FUNCTION_BLOCK FB_PrintModule_WEU EXTENDS FB_PrintModule_Base
VAR_INPUT
  fPUPlate1_Temperature : LREAL;  // PU Plate1 temperature
  fPUPlate2_Temperature : LREAL;  // PU Plate2 temperature
END_VAR
VAR
  (* Module specific sub-modules - WEU module contains a 
    - print position (encoder input to print domain translation)
    - Mark sensor with a mark detection module which provices a camera trigger and start position detection
    - Mark definition (used by the detection and camera)
  *)
  fbPrintPosition    : FB_PrintPositionDmax;   // a position per pm (external encoder wheel)
  fbMarkCameraWeu    : FB_MarkCamera_WEU;      // Mark detection camera
  
  // sync CT trigger with Camera detection
  _bNewCT             : BOOL;   // a new ct is received to be treated
  _iNewCT             : I_CT;   // new ct to be treated
  _bNewStartPosX0     : BOOL;   // a new startpos detected by cam
  _nNewStartPosX0     : DINT;   // new startpos X0 deteced by cam
  
  fbEncoderResoDetect : FB_EffectiveEncoderResolutionDetection;     // Effective encoder resolution detection
  fbFineAlignement    : FB_FineAlignement;     // additional grid corrections, PU Deformation/correction (4p, banana, ...)

  // messages specific
  fbMsgWeu            : ARRAY[1..nC_NumMsgWeu] OF FB_MESSAGE;  (*Messages*)
  
  // view
  fbView              : FB_PrintModule_WEU_View;    // additional controls for print module visus
END_VAR
VAR CONSTANT
  nC_NumMsgWeu        : UDINT := 6;           // number of internal messages
END_VAR

IF NOT bInit THEN RETURN; END_IF

// position
fbPrintPosition.fEnoderResolution := _pModuleMachineState^.fEncoderResolution;    // encoder resolution from machine
fbPrintPosition();

// -------------------------
// StartTrigger evaluation -> apply new CT to Tracking (created from CTM externally)
// Synchronize CT (EvPos) received from CTManger (Main) to the local StartTrigger detection and positioning
// -- reset triggers if not active
IF NOT bReadyForPrinting THEN
  _bNewCT := 0; _bNewStartPosX0 := 0;
END_IF
// -- new StartTrigger (X0)
IF bReadyForPrinting AND _iStartPos.bStartTrig AND _iStartPos.bValid THEN
  // buffer/save new start trigger
  _bNewStartPosX0 := TRUE;
  _nNewStartPosX0 := _iStartPos.nStartPositionX0;      // save detected start position for next CT to be applied to this module¨
  
  LogLvl(Lvl:=E_LogSeverity.Debug, Msg:=F_Concat3(
    F_Concat2(_pModuleSetup^.aName, ' New StartTrigger detected:'),
    F_Concat2(' at position X0:', TO_STRING(_nNewStartPosX0)),
    F_Concat2(' PM is now at: ', TO_STRING(fbPrintPosition.getPosition())),
  ));
  
  IF _bNewCT THEN   // we have an attached CT
      LogLvl(Lvl:=E_LogSeverity.Debug, Msg:=F_Concat3(
      F_Concat2(_pModuleSetup^.aName, ' Track NewCT:'),
      F_Concat2(' internal (print)Pos X0:', TO_STRING(_nNewStartPosX0)),
      F_Concat2(' with CT:', _iNewCT.print(0))
    ));
    
    _iNewCT.nPosPrint_X0 := _nNewStartPosX0;                        // set print pos to new dected in this module position domain
    fbCTTracker.RegisterCT(iCT:=_iNewCT, nX0:=_nNewStartPosX0);     // register ct for tracking in modules position and tracking system
  ELSE
    // spurious trigger (CTs not yet arrived at PMx, but receive some StartTriggers
    LogLvl(Lvl:=E_LogSeverity.Debug, Msg:=F_Concat3('StartTrigger at Pos X0:', TO_STRING(_nNewStartPosX0), ' but no CT received'));
	END_IF
  
  // reset internals (saved triggers)
  _bNewCT := FALSE; _iNewCT := 0; 
  _bNewStartPosX0 := FALSE;
END_IF

// Camera (is per module)
fbMarkCameraWeu(
  bReadyForPrinting   := bReadyForPrinting,
  nCurrentPosition    := _iPrintPosition.getPosition(),
  fCurrentSpeed       :=_iPrintPosition.getSpeed(),
  bPrintMarkExist     :=_pModuleMachineState^.bPrintMarkExist,
  bPrintDirReverse    :=_pModuleMachineState^.bPrintDirection,
  nUsePerRepeatInLine :=SEL(_pModuleMachineState^.nUsePerRepeatInLine=0, _pModuleMachineState^.nUsePerRepeatInLine, 1),
  fMarkSizeDefault    :=_pModuleMachineState^.fMarkBaseSize,
  fMarkDistRepeatToStartMark := _pModuleMachineState^.fMarkDistToStartMark,
  fMarkDistFromCenter := _pModuleMachineState^.fMarkToPrintdataCenterY
);

// Effective Encoder detection - Neutral fibre calculation with additional mark sensors
fbEncoderResoDetect(
  //bIKp_MarkTrigger01:=,
  //tIKp_TimeStampPos01:=,
  //tIKn_TimeStampNeg01:=,
  //bIKp_MarkTrigger02:=,
  //tIKp_TimeStampPos02:=,
  //tIKn_TimeStampNeg02:=,
  nPulse:=TO_DINT(fbPrintPosition.IlEncoderPulse),
  fCurrentResolution:=_pModuleMachineState^.fEncoderResolution,
  fEncoderPulseDistMin:=_pModuleMachineState^.fEncoderDetectPulseMin,
  fEncoderPulseDistMax:=_pModuleMachineState^.fEncoderDetectPulseMax,
  nDisInPulseFilterSz:=_pModuleMachineState^.nEncoderDetectFilterSz,
  fMinMarkLength:=(0.5 - 0.1) * _pModuleMachineState^.fMarkBaseSize * 1_000_000,  // 0.5*a (0*a from triangle)
  fMaxMarkLength:=(  3 + 0.1) * _pModuleMachineState^.fMarkBaseSize * 1_000_000,  //   2*a (1*a from triangle) 
  // --> the following would only work when teached
  //fMinMarkLength:=fbMarkCameraWeu.pFbMarkDefinition^.fMinMarkLength - fbMarkCameraWeu.pFbMarkDefinition^.fMarkLengthMargin * 1_000_000,
  //fMaxMarkLength:=fbMarkCameraWeu.pFbMarkDefinition^.fMaxMarkLength + fbMarkCameraWeu.pFbMarkDefinition^.fMarkLengthMargin * 1_000_000,
  //bUpdate=>,
  fDisInPulse=>_pModuleMachineFeedback^.fEncoderStepsMeasured
);

(*PU corrections*)
IF GVL_Deformation.bC_UsePUDeformation THEN
  fbFineAlignement.fT_PL1 := fPUPlate1_Temperature;
  fbFineAlignement.fT_PL2 := fPUPlate2_Temperature;
  fbFineAlignement();
END_IF

fbView();

// call module base
SUPER^();

// messages print module
fbMsgWeu[ 1](bI_Status := bTestMsg OR fbMarkCameraWeu.bMissingMarks);
fbMsgWeu[ 2](bI_Status := bTestMsg OR _pModuleMachineState^.bDriftControlMissMarks);
fbMsgWeu[ 3](bI_Status := bTestMsg OR fbMarkCameraWeu.bMarkDetectionErrors);
fbMsgWeu[ 4](bI_Status := bTestMsg OR fbMarkCameraWeu.bTeachError);
fbMsgWeu[ 5](bI_Status := bTestMsg OR fbMarkCameraWeu.bImageLengthInvalid);
fbMsgWeu[ 6](bI_Status := bTestMsg OR _bGridLimited);

IF fb_MsgQueue.bO_ReceiptMessage THEN
  fbMarkCameraWeu.ackErrors();
  _bGridLimited := FALSE;
END_IF

// simulation
SimUpdate();

PROPERTY bForceNoCorrectionButYShiftMode : BOOL
SET
FOR nCtr := 1 TO GVL_WEU.nC_MaxWorkerPrintPerPm DO
  fbWorkerPrint[nCtr].bForceNoCorrectionButShiftMode := bForceNoCorrectionButYShiftMode;
END_FOR
END_SET
END_PROPERTY

METHOD Init : BOOL
VAR_INPUT
  pModulesSetup         : POINTER TO ST_CassetteSetup;          // Module Setup Settings
  pAdsSa                : POINTER TO FB_ADS_DVTSHEETALIGNMENT;  // ADS sheet alignement
  pAdsCam               : POINTER TO FB_ADS_CAMERA;             // ADS camera
  pAdsParent            : POINTER TO FB_ADS_Config;             // Parent ADS config reference (Parent ADS block and module ref)

  // config print
  fCycleTime            : LREAL;                // task cycle time in [s]
  fPrintUnitWidth       : LREAL;                // PrintUnit width mechanical [m]
  // references
  iModule               : I_Module;             // system status interface (for sleep, estop, ...), may shadow states from machine inputs
  iPrintGlobal          : I_PrintGlobal;        // interface for module to master (main) communication
  pMachineInputs        : POINTER TO ST_ModuleMachineInterface_IN;
  pMachineOutputs       : POINTER TO ST_ModuleMachineInterface_OUT;
END_VAR
VAR
  nCtr : UDINT;
END_VAR
// Parameter checks
IF pModulesSetup = 0 OR pAdsSa = 0 OR pAdsCam = 0 OR 
    pMachineInputs = 0 OR pMachineOutputs = 0 THEN
    // set here from local fb instances: OR iModuleMaster = 0 OR iPosition = 0 OR iStartPos = 0 THEN
  LogError('init(): Invalid parameter');
  RETURN;
END_IF

// position
fbPrintPosition.Init(fPrintResolution:=pModulesSetup^.pSetupPrint^.nPrintResolution, fSubPxResolution:=pModulesSetup^.pSetupPrint^.nSubPixelResolution, fTaskCycleTime:=fCycleTime);
_iPrintPosition := fbPrintPosition;  // select reference position

// -- Mark camera
fbMarkCameraWeu.InitMarkCamera(
  fPrintUnitResolution:=_iPrintPosition.fPrintResolution, 
  fPrintUnitSubPx:=_iPrintPosition.fSubPxResolution
);
fbMarkCameraWeu.sVisuName := 'VISU_MarkCamera_WEU';
fbWorkerCamera.RegisterCamera(fbMarkCameraWeu);

// -- Sheet/Camera trigger & mark detection
_iStartPos := fbMarkCameraWeu.fbMarkDetection;  // select start position detection

SUPER^.Init(
  pModulesSetup     := pModulesSetup,
  pAdsSa            := pAdsSa,
  pAdsCam           := pAdsCam,
  pAdsParent        := pAdsParent,
  // config print
  fCycleTime        := fCycleTime,
  fPrintUnitWidth   := fPrintUnitWidth,
  // references     
  iPrintGlobal      := iPrintGlobal,     // internal subm
  iModule           := iModule, 
  pMachineInputs    := pMachineInputs,
  pMachineOutputs   := pMachineOutputs
);

// Effective Encoder Resolution detection (NeutralFibre correction)
fbEncoderResoDetect.Init();

// additional grid point corrections
fbFineAlignement.init(pAdsCam := pAdsCam, fPxReso := _iPrintPosition.fPrintResolution, fPuWidth := fPrintUnitWidth);
// - register them to workers
FOR nCtr := 1 TO GVL_WEU.nC_MaxWorkerPrintPerPm DO
  fbWorkerPrint[nCtr].RegisterGridCorrection(iGridCorrection:=fbFineAlignement);
END_FOR 

fbView.init(pModule:=THIS, pPositioning:=ADR(fbPrintPosition));
setLogLevels(lvl:=E_LogSeverity.Info);

FOR nCtr := 1 TO nC_NumMsgWeu DO
  fbMsgWeu[nCtr].pI_MsgConfig       := ADR(sL_MsgConfig);
  fbMsgWeu[nCtr].iI_MsgLocation     := 1;
END_FOR;
fbMsgWeu[ 1].iI_MsgNumber      := eCPr_PrintMarkError_Generic;        // mark detection error
fbMsgWeu[ 2].iI_MsgNumber      := eCMa_DRIFT_CONTR_ERROR;             // drift controller error
fbMsgWeu[ 3].iI_MsgNumber      := eCPr_SHEET_MARK_DETECTION;          // mark error missing/faulty
fbMsgWeu[ 4].iI_MsgNumber      := eC_STAG_CAM_TEACH_ERROR;            // teach error
fbMsgWeu[ 5].iI_MsgNumber      := eC_STAG_IMAGELENGTH_NOT_SUPPORTED;  // image length not supported (out of supported range)
fbMsgWeu[ 6].iI_MsgNumber      := eC_STAG_DEFORMATION_LIMITED;        // deformation calculated was limited to min/max before sending

Init := bInit;   // set in the SUPER class
END_METHOD

PROPERTY pMsgConfig : POINTER TO ST_MSG_CONFIG
GET
pMsgConfig := ADR(sL_MsgConfig);
END_GET
END_PROPERTY

METHOD PROTECTED setLogLevels
VAR_INPUT
  lvl : E_LogSeverity;
END_VAR
// - fb itself
LogLevel := lvl;
// - base
SUPER^.setLogLevels(lvl:=lvl);
// - weu
fbPrintPosition.LogLevel := lvl;
fbMarkCameraWeu.LogLevel := lvl;
END_METHOD

METHOD PRIVATE SimUpdate
VAR_INPUT
END_VAR
VAR_INST
  rfTrig_SimEnable : RF_TRIG;
  
  //parameter backup
  fCamMark_ToPrint, fCamMark_toDetect : LREAL;
  fCamNo_ToPrint, fCamNo_toDetect : LREAL;
END_VAR
rfTrig_SimEnable(CLK:=fbSim.bSimEnable);
IF    rfTrig_SimEnable.RT THEN
  // ev. enable
  //fbWorkerCamera.bWorkerEnable := TRUE;
  //fbWorkerDeformation.bWorkerEnable := TRUE;
  //fbWorkerPrint[1].bWorkerEnable := TRUE;
  //fbWorkerPrint[2].bWorkerEnable := TRUE;
  
  fbPrintPosition.bSimEnable  := TRUE;
  fbMarkCameraWeu.bSimulate := TRUE;

  // set some working config values
  // -backup original
  fCamMark_ToPrint  := fbMarkCameraWeu.fCameraToPrintOffset;
  fCamMark_toDetect := fbMarkCameraWeu.fDetectToCameraOffset;
  // -set sim val
  fbMarkCameraWeu.fCameraToPrintOffset := 0.4;
  fbMarkCameraWeu.fDetectToCameraOffset := 0.01;
  
  
ELSIF rfTrig_SimEnable.FT THEN
  // ev. disable
  fbPrintPosition.bSimEnable  := FALSE;
  fbMarkCameraWeu.bSimulate := FALSE;

  fbMarkCameraWeu.fCameraToPrintOffset := fCamMark_ToPrint;
  fbMarkCameraWeu.fDetectToCameraOffset := fCamMark_toDetect;
  
ELSIF fbSim.bSimEnable THEN
  // enabled
  ;
ELSE
  ; // disabled
END_IF
END_METHOD

(*
  Container triggered at position - callback.
*)
METHOD trigger : BOOL
VAR_INPUT
	sEvPos	: ST_PositionEventData;
END_VAR
IF NOT bInit THEN RETURN; END_IF
IF sEvPos.iCT = 0 THEN RETURN; END_IF


// buffer new ct
_bNewCT := TRUE;
_iNewCT := sEvPos.iCT;

LogLvl(Lvl:=E_LogSeverity.Debug, Msg:=F_Concat3(
  F_Concat2(_pModuleSetup^.aName, ' NewCT PosEv:'),
  F_Concat2(' at (Main)TrackPos:', TO_STRING(sEvPos.nTrigPos)),
  F_Concat2(' with CT:', sEvPos.iCT.print(0))
));
END_METHOD

END_FUNCTION_BLOCK

(* stored: Version 1.1.0.1, ProductVersion 3.1.4024.11
   POU FB_PrintModule_WEU: Id {bf81d19f-9fa7-4acb-8cca-087a288b3f4d}, SpecialFunc None
   Folder I_PositionEvent_ovrd: Id {212612fd-c98f-4fcb-8ea9-fac5585d1647}
   Folder Simulation: Id {ff45cf45-269f-4fec-ab1d-0aca9951a18d}
   Property bForceNoCorrectionButYShiftMode: Id {b65a9350-831c-45ea-8f78-0fa9026ef73e}
   Set Set: Id {3d096227-cb0c-4e6c-ae20-0ca9a6fd3412}
   Method Init: Id {fba0a279-e9f9-46b1-8f8f-0e7a0e308a34}
   Property pMsgConfig: Id {3f9ad2f8-f49c-46e8-8c7b-162fe18749a6}
   Get Get: Id {5bcaf950-0c98-4a16-8209-bb10ff6fbca0}
   Method setLogLevels: Id {e26383c7-5f29-468c-b845-4944132a7335}
   Method SimUpdate: Id {86d331a7-7239-49bc-b197-44cccc5c4107}
   Method trigger: Id {a0aceb5d-071c-4ce1-a837-1712d7194423} *)
